// TIA Portal project "Lab6Exp1" (V16)

(* hardware
DEVICE "S7300/ET200M station_1"  S7-300 station
   slot 0: "Rail_0"  Rail  6ES7 390-1***0-0AA0
   slot 2: "PLC_1"  CPU 315-2 PN/DP  6ES7 315-2EH14-0AB0  V3.2
      slot 2: "PROFINET interface_1"  PN-IO
         slot 1: "Port_1"  Port
         slot 2: "Port_2"  Port
*)

// ===== PLC "PLC_1"  CPU 315-2 PN/DP =====

VAR_GLOBAL   // PLC tag table "Default tag table"
   "Tag_1" AT %C10 : Counter;
   "Tag_2" AT %I1.0 : Bool;
   "Tag_3" AT %I1.1 : Bool;
   "Tag_4" AT %I1.2 : Bool;
   "Tag_5" AT %MW10 : Word;
   "Tag_6" AT %MW12 : Word;
   "Tag_7" AT %Q1.0 : Bool;
   "Tag_8" AT %I2.0 : Bool;
   "Tag_9" AT %I2.1 : Bool;
   "Tag_10" AT %I2.2 : Bool;
   "Tag_11" AT %C11 : Counter;
   "Tag_12" AT %Q2.0 : Bool;
   "Tag_13" AT %MW20 : Word;
   "Tag_14" AT %MW22 : Word;
   "Tag_15" AT %C12 : Counter;
   "Tag_16" AT %I3.0 : Bool;
   "Tag_17" AT %I3.1 : Bool;
   "Tag_18" AT %I3.2 : Bool;
   "Tag_19" AT %I3.3 : Bool;
   "Tag_20" AT %Q3.0 : Bool;
   "Tag_21" AT %MW30 : Word;
   "Tag_22" AT %MW31 : Word;
   "Tag_23" AT %MW32 : Word;
   "Tag_24" AT %I4.0 : Bool;
   "Tag_25" AT %C13 : Counter;
   "Tag_26" AT %MW40 : Word;
   "Tag_27" AT %I4.1 : Bool;
   "Tag_28" AT %I4.2 : Bool;
   "Tag_29" AT %C14 : Counter;
   "Tag_30" AT %MW42 : Word;
   "Tag_31" AT %MW44 : Int;
   "Tag_32" AT %MW46 : Int;
   "Tag_33" AT %I0.0 : Bool;
   "Tag_34" AT %I0.1 : Bool;
   "Tag_35" AT %M0.0 : Bool;
   "Tag_36" AT %C1 : Counter;
   "Tag_37" AT %Q0.0 : Bool;
   "Tag_38" AT %C2 : Counter;
END_VAR

ORGANIZATION_BLOCK "Main"   // OB1, LAD
TITLE = "Main Program Sweep (Cycle)"
{ S7_Optimized_Access := 'FALSE' }
VERSION : 0.1
   VAR_TEMP
      OB1_EV_CLASS : Byte;   // Bits 0-3 = 1 (Coming event), Bits 4-7 = 1 (Event class 1)
      OB1_SCAN_1 : Byte;   // 1 (Cold restart scan 1 of OB 1), 3 (Scan 2-n of OB 1)
      OB1_PRIORITY : Byte;   // Priority of OB Execution
      OB1_OB_NUMBR : Byte;   // 1 (Organization block 1, OB1)
      OB1_RESERVED_1 : Byte;   // Reserved for system
      OB1_RESERVED_2 : Byte;   // Reserved for system
      OB1_PREV_CYCLE : Int;   // Cycle time of previous OB1 scan (milliseconds)
      OB1_MIN_CYCLE : Int;   // Minimum cycle time of OB1 (milliseconds)
      OB1_MAX_CYCLE : Int;   // Maximum cycle time of OB1 (milliseconds)
      OB1_DATE_TIME : Date_And_Time;   // Date and time OB1 started
   END_VAR
   VAR_TEMP   // added for the SCL form of the ladder/FBD networks
      _w1 : Bool;
   END_VAR
BEGIN

REGION Network 1: Testing a Counter C10:Counting up only
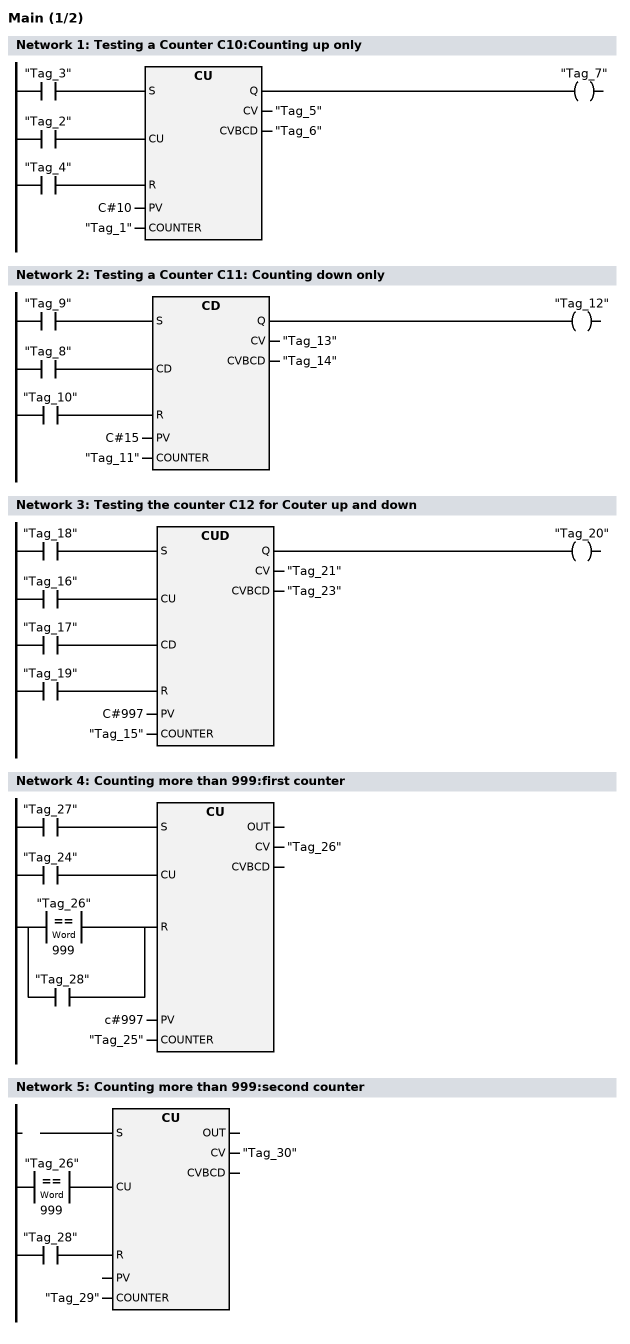
   // no SCL statement known for Cu: written as a call
   Cu(cu := "Tag_2",
      s := "Tag_3",
      r := "Tag_4",
      pv := C#10,
      "counter" := "Tag_1",
      q => #_w1,
      cv => "Tag_5",
      cvbcd => "Tag_6");
   "Tag_7" := #_w1;
END_REGION

REGION Network 2: Testing a Counter C11: Counting down only
   // no SCL statement known for Cd: written as a call
   Cd(cd := "Tag_8",
      s := "Tag_9",
      r := "Tag_10",
      pv := C#15,
      "counter" := "Tag_11",
      q => #_w1,
      cv => "Tag_13",
      cvbcd => "Tag_14");
   "Tag_12" := #_w1;
END_REGION

REGION Network 3: Testing the counter C12 for Couter up and down
   // no SCL statement known for Cud: written as a call
   Cud(cu := "Tag_16",
       cd := "Tag_17",
       s := "Tag_18",
       r := "Tag_19",
       pv := C#997,
       "counter" := "Tag_15",
       q => #_w1,
       cv => "Tag_21",
       cvbcd => "Tag_23");
   "Tag_20" := #_w1;
END_REGION

REGION Network 4: Counting more than 999:first counter
   // no SCL statement known for Cu: written as a call
   Cu(cu := "Tag_24",
      s := "Tag_27",
      r := ("Tag_26" = 999) OR "Tag_28",
      pv := c#997,
      "counter" := "Tag_25",
      cv => "Tag_26");
END_REGION

REGION Network 5: Counting more than 999:second counter
   // no SCL statement known for Cu: written as a call
   Cu(cu := "Tag_26" = 999, r := "Tag_28", "counter" := "Tag_29", cv => "Tag_30");
END_REGION

REGION Network 6: Counting more than 999:final Result
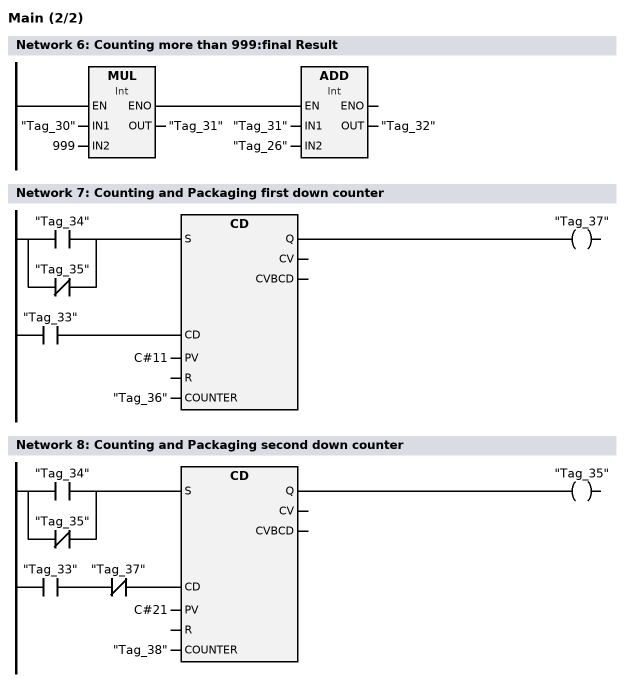
   RUNG wire#powerrail
      { S7_Templates := "SrcType := Int"; S7_GenerateENO := "TRUE" } Mul(in1 := "Tag_30", in2 := 999, out => "Tag_31")
      { S7_Templates := "SrcType := Int"; S7_GenerateENO := "TRUE" } Add(in1 := "Tag_31", in2 := "Tag_26", out => "Tag_32")
   END_RUNG
   // the same network as SCL:
   // ENO of a box is taken as its EN; it also drops when the box reports an error
   "Tag_31" := "Tag_30" * 999;
   "Tag_32" := "Tag_31" + "Tag_26";
END_REGION

REGION Network 7: Counting and Packaging first down counter
   // no SCL statement known for Cd: written as a call
   Cd(cd := "Tag_33", s := "Tag_34" OR NOT "Tag_35", pv := C#11, "counter" := "Tag_36", q => #_w1);
   "Tag_37" := #_w1;
END_REGION

REGION Network 8: Counting and Packaging second down counter
   // no SCL statement known for Cd: written as a call
   Cd(cd := "Tag_33" AND NOT "Tag_37",
      s := "Tag_34" OR NOT "Tag_35",
      pv := C#21,
      "counter" := "Tag_38",
      q => #_w1);
   "Tag_35" := #_w1;
END_REGION
END_ORGANIZATION_BLOCK